FUNCTION_BLOCK Motor IMPLEMENTS IDevice
VAR_INPUT
END_VAR
VAR_OUTPUT
END_VAR
VAR
	isOn : BOOL := FALSE;       
END_VAR

METHOD PUBLIC turnOn
VAR_INPUT
END_VAR
isOn := true;
END_METHOD

END_FUNCTION_BLOCK

(* stored: Version 1.1.0.1, ProductVersion 3.1.4024.11
   POU Motor: Id {dbe739ed-a399-46b1-8792-527b21aebda7}, SpecialFunc None
   Method turnOn: Id {6f161a4f-8a82-4c99-be1f-28c3318f397c} *)
